// TIA Portal V20 export
TYPE "UDT_ConfigDesPaletizador"
   STRUCT
      VeloManual : Int := 1000;   // Velocidad en Manual
      VeloCapa : Int := 2000;   // Velocidad de Movimiento de Capa
      VeloRapidaDown : Int := 8000;   // Velocidad Rapida de Movimiento Down
      VeloLentaDown : Int := 3000;   // Velocidad Lenta de Movimiento Down
      VeloRapidaUp : Int := 8000;   // Velocidad Rapida de Movimiento Up
      VeloLentaUp : Int := 2000;   // Velocidad Lenta de Movimiento Up
      PosVeloLentaDown : Int := 500;   // Posicion al final para entrada en Lenta en MOv. Down
      PosVeloLentaUp : Int := 500;   // Posicion al final para entrada en Lenta en MOv. Up
      AlturaMax : Int := 4700;   // Altura MAx de Posicion del elevador
      AlturaMin : Int := 200;   // Altura Min de Posicion del Elevador
      AlturaPaleta : Int := 165;   // Altura de Paleta
      AlturaGalibo : Int := 3660;   // Altura de Control de Mov al Puesto
      AlturaSensoresGalibo : Int := 3660;   // Altura de Control de Mov al Puesto
      AlturaBarrera : Int := 3900;   // Altura de la Paleta en el Nivel (Dinamico)
      PosicionCarga : Int := 805;   // Altura de Carga de Paleta
      PosicionDesCarga : Int := 225;   // Altura de DesCarga de Paleta
   END_STRUCT;
END_TYPE
